//---------------------------------------------------------------------------------------------------------------
//
//  HAUD 2024.12.19
//
//
//  fb_SenderBuffer
//  - inherits fb_Instance, which provides a design pattern in order to build different specific processes in a structured way
//  - uses 1 XtsStation via _ItfProcessCollector
//  - used for targeting movers to predetermined substation of process control (one to one)
//  - processes are connected via linked list
//    - entry in list is detected
//    - entry in list determines count and place of used XtsStations in target process
//
//
//  - constructed with fb_Instance main state (_eState) in addition to a substate (_eStateProgress)
//  - substate enables to handle procedures within main state by preventing race conditions 
//    with the help of small steps and decisions with clear separation from each other 
//
//---------------------------------------------------------------------------------------------------------------//
// This SOFTWARE is provided as an Exemple by THE PROVIDER "as is" and "with all faults." THE PROVIDER makes no  //
// representations or warranties of any kind concerning the safety, suitability, lack of viruses, inaccuracies,  //
// typographical errors, or other harmful components of this SOFTWARE. There are inherent dangers in the use of  //
// any software, and you are solely responsible for determining whether this SOFTWARE is compatible with your    //
// equipment and other software installed on your equipment. You are also solely responsible for the protection  //
// of your equipment and backup of your data, and THE PROVIDER will not be liable for any damages you may suffer //
// in connection with using, modifying, or distributing this SOFTWARE.                                           //
//---------------------------------------------------------------------------------------------------------------//
FUNCTION_BLOCK fb_SenderBuffer EXTENDS fb_Instance
VAR
  _nProcessTarget               : E_INSTANCE;     // who am I connected to

  // target XTS station range
  _nTargetStationLast           : UINT;           // where does the target process end
  _nTargetStationFirst          : UINT;           // where does the target process start

  _rCheckPos                    : LREAL;

  _WriteResult                  : ST_PROCESS_LIST_RESULT;   // last job written to target
  _DeleteResult                 : ST_PROCESS_LIST_RESULT;   // last job executed

  _idx                          : UINT;
  _nTargetIndex                 : ARRAY[1..SIZEOF(T_PROCESS)*8] OF USINT; // helper var to copy to my process (_ItfProcessCollector[_nProcess].TargetIndex)

  _MoverInfo                    : ST_MOVER_INFO;      // Information from the Mover in Station
  _StationState                 : ST_STATION_STATE;   // fb_SenderBufferInfeed has only one XtsStation to work

  _nBatch                       : udint;
END_VAR

//-----------------------------------------------------------------------------
//-----------------------------------------------------------------------------
// check pointer and interface
// connect Ctrl/State to _ItfProcessCollector
// set message device identification
//-----------------------------------------------------------------------------
IF NOT Check() THEN 
  RETURN; 
END_IF
//-----------------------------------------------------------------------------
// check init command (hard reset)
//-----------------------------------------------------------------------------
_eCmd                                 := _InstanceCtrl[_nProcess].Cmd;
IF (_eCmd <> _eCmdOld)
THEN
  CASE _eCmd
  OF
    E_INSTANCE_CMD.INIT:
      // clear init info
      _nBatch                         := 0;
      _eInit                          := _ItfProcessCollector[_nProcess].Init(FALSE);
  
      IF _ItfProcessList[_nProcess].InitList()  // clear linked list
      THEN
        Clear();
        _eStateInstance               := E_INSTANCE_STATE.INIT;
        _eStateProgress               := E_PROGRESS.PROGRESS_INIT;
      END_IF

    E_INSTANCE_CMD.CLEAR:
        _eStateInstance               := E_INSTANCE_STATE.DISABLED;
        _eStateProgress               := E_PROGRESS.PROGRESS_INIT;
  END_CASE
  CmdLog();
  _eCmdOld                            := _eCmd;
END_IF
//-----------------------------------------------------------------------------
// cyclic information of mover and station
//-----------------------------------------------------------------------------
_StationState                         := _ItfProcessCollector[_nProcess].GetStationState  (_ItfProcessCollector[_nProcess].StationLast);
_MoverInfo                            := _ItfProcessCollector[_nProcess].GetMoverInStation(_ItfProcessCollector[_nProcess].StationLast);
//-----------------------------------------------------------------------------
//-----------------------------------------------------------------------------
// state machine for buffer to OutputR1 and OutputR2
//-----------------------------------------------------------------------------
CASE _eStateInstance // main state machine
OF
  E_INSTANCE_STATE.NULL:           // first cycle init
    IF _ItfProcessList[_nProcess].InitList()
    THEN
      _eInit                          := _ItfProcessCollector[_nProcess].Init(FALSE);
      _eStateProgress                 := E_PROGRESS.PROGRESS_INIT;
      _eStateInstance                 := E_INSTANCE_STATE.INIT;
    END_IF


  E_INSTANCE_STATE.INIT:              // plausibility checks and _ItfProcessCollector Init
    //-------------------------------------------------------------------------
    CASE _eStateProgress
    OF
    //-------------------------------------------------------------------------
      E_PROGRESS.PROGRESS_ERROR:
        IF (_nProcessTarget > 0) AND
           (_nProcessTarget < E_INSTANCE.INSTANCE_MAX)
        THEN
          _eStateProgress             := E_PROGRESS.PROGRESS_INIT;
        END_IF

    // E_INSTANCE_STATE.INIT:
    //-------------------------------------------------------------------------
      E_PROGRESS.PROGRESS_INIT:
        IF NOT (_nProcessTarget > 0) OR
           NOT (_nProcessTarget < E_INSTANCE.INSTANCE_MAX)
        THEN
          // an invalid target you must have not
          _eStateProgress             := E_PROGRESS.PROGRESS_ERROR;
        ELSE
          _eStateProgress             := E_PROGRESS.PROGRESS_BUSY;
        END_IF

    // E_INSTANCE_STATE.INIT:
    //-------------------------------------------------------------------------
      E_PROGRESS.PROGRESS_BUSY:
        // wait for my process collector check (_State.Check) to be done
        //  - checks range of XtsStations
        //  - checks count of XtsStations
        IF (_State.Check = E_PROCESS_CHECK.PROCESS_CHECK_DONE)
        THEN
          _eInit                      := _ItfProcessCollector[_nProcess].Init(TRUE);
  
          IF (_eInit = E_PROGRESS.PROGRESS_DONE)
          THEN
            IF NOT (_nProcessTarget > 0) OR
               NOT (_nProcessTarget < E_INSTANCE.INSTANCE_MAX)
            THEN
              // an invalid target you must have not
              _eStateProgress         := E_PROGRESS.PROGRESS_ERROR;

              _stMsg.eType            := E_MessageType.eMessageError;
              _stMsg.eSubdevice       := e_Subdevice.Instance_BufferOutfeed;
              _stMsg.iErrorNumber     := _nProcessTarget;
              _stMsg.sText            := concat(TO_STRING(_eStateInstance), ': ProcessTarget: ');
              _stMsg.sText            := concat(_stMsg.sText, TO_STRING(_eStateProgress));
              f_MessageSet(_stMsg);

            ELSE
              _nTargetStationLast     := _ItfProcessCollector[_nProcessTarget].StationLast;
              _nTargetStationFirst    := _ItfProcessCollector[_nProcessTarget].StationFirst;

              // initialization of Infeed: _ItfProcessCollector with XtsStation
              _Ctrl.Cmd               := E_PROCESS_CTRL.PROCESS_DISABLE;  // first, switch off _ItfProcessCollector and XtsStation
              _eStateProgress         := E_PROGRESS.PROGRESS_INIT;        // clear sub state
              _eStateInstance         := E_INSTANCE_STATE.DISABLED;       // switch to disabled as default after startup
            END_IF
          END_IF
        END_IF
    END_CASE
END_CASE
//-----------------------------------------------------------------------------
//-----------------------------------------------------------------------------
// DISABLED:
//  - clear local list result data
//  - wait for enable from the outside
//  - wait for an entry in my list
//-----------------------------------------------------------------------------
CASE _eStateInstance
OF
  E_INSTANCE_STATE.DISABLED:
    //-------------------------------------------------------------------------
    CASE _eStateProgress
    OF
      E_PROGRESS.PROGRESS_INIT:
        _eStateProgress               := E_PROGRESS.PROGRESS_BUSY;
        // clear data for a new round
        memset(ADR(_ListResult), 0, SIZEOF(_ListResult));

        _Ctrl.ActivateStation         := 0;
        _Ctrl.NestMask                := 1;
        
    // E_INSTANCE_STATE.DISABLED:
    //-------------------------------------------------------------------------
      E_PROGRESS.PROGRESS_BUSY:
        CASE _eCmd
        OF
          E_INSTANCE_CMD.ENABLE:      // turn it on!!
            _eStateInstance           := E_INSTANCE_STATE.DETECTION;
            _eStateProgress           := E_PROGRESS.PROGRESS_BUSY;

  
            IF (_MessageLevel > E_MessageType.eMessageInfo)
            THEN
              _stMsg.eType            := E_MessageType.eMessageVerbose;
              _stMsg.eSubdevice       := e_Subdevice.Instance_Sender_Buffer;
              _stMsg.iErrorNumber     := 0;
              _stMsg.sText            := concat(TO_STRING(_eStateInstance), ': ');
              _stMsg.sText            := concat(_stMsg.sText, TO_STRING(_eStateProgress));
              f_MessageSet(_stMsg);
            END_IF
        END_CASE
    END_CASE
END_CASE
//-----------------------------------------------------------------------------
// DETECTION: 
//  - check inked list and GetHead()
//  - copy job data
//  - switch on process
//-----------------------------------------------------------------------------
CASE _eStateInstance
OF
  E_INSTANCE_STATE.DETECTION:
    //-------------------------------------------------------------------------
    CASE _eStateProgress
    OF
      E_PROGRESS.PROGRESS_INIT:
        IF (_eCmd = E_INSTANCE_CMD.PROCEED)
        THEN
          _eStateProgress             := E_PROGRESS.PROGRESS_BUSY;
        END_IF
    END_CASE
    // E_INSTANCE_STATE.DETECTION
    //-------------------------------------------------------------------------
    CASE _eStateProgress
    OF
      E_PROGRESS.PROGRESS_BUSY:
        IF (_eCmd = E_INSTANCE_CMD.DISABLE)
        THEN
          _eStateInstance             := E_INSTANCE_STATE.DISABLED;
          _eStateProgress             := E_PROGRESS.PROGRESS_INIT;

        ELSIF (_ItfProcessList[_nProcess].Count > 0)
        THEN
          // get new job order for my process
          // check my list for a new round of movers
          _ListResult                 := _ItfProcessList[_nProcess].GetHead();  // the list results carries information about the requirements of the target process (who and where)

          IF (_ListResult.wState <> 0)
          THEN
            // error in list results must not appear
            // if you land here, there is somethng wrong with the initialization or configuration of the linked list
            _eStateProgress           := E_PROGRESS.PROGRESS_ERROR;

            _stMsg.eType              := E_MessageType.eMessageError;
            _stMsg.eSubdevice         := e_Subdevice.Process_LinkedList_GetHead;
            _stMsg.iErrorNumber       := _ListResult.wState;
            _stMsg.sText              := concat(TO_STRING(_eStateInstance), ': ');
            _stMsg.sText              := concat(_stMsg.sText, TO_STRING(_eStateProgress));
            f_MessageSet(_stMsg);

          ELSE
            IF (_MessageLevel > E_MessageType.eMessageError)
            THEN
              _stMsg.eType            := E_MessageType.eMessageInfo;
              _stMsg.eSubdevice       := e_Subdevice.Process_LinkedList_GetHead;
              _stMsg.iErrorNumber     := 0;
              _stMsg.sText            := concat(TO_STRING(_eStateInstance), ': ');
              _stMsg.sText            := concat(_stMsg.sText, '_ListResult.stData.wTarget: ');
              _stMsg.sText            := concat(_stMsg.sText, _ItfProcessCollector[_nProcess].BitsToString(_ListResult.stData.wTarget));
              f_MessageSet(_stMsg);
            END_IF

            _ProcessData              := _ListResult.stData;  // list result contains data for target process

            IF NOT (_ProcessData.wTarget > 0)
            THEN
              // no data, no cry
              _DeleteResult           := _ItfProcessList[_nProcess].RemoveHeadValue();
            ELSE
              _eStateProgress         := E_PROGRESS.PROGRESS_CHECK;

              IF (_MessageLevel > E_MessageType.eMessageEmpty)
              THEN
                _stMsg.eType            := E_MessageType.eMessageBatch;
                _stMsg.eSubdevice       := e_Subdevice.Instance_Sender_Buffer;
                _stMsg.iErrorNumber     := _ProcessData.wTarget;
                _stMsg.sText            := concat('_ProcessData.wTarget: ', _ItfProcessCollector[_nProcess].BitsToString(_ProcessData.wTarget));
                _stMsg.sText            := concat(_stMsg.sText, ': ');
                _stMsg.sText            := concat(_stMsg.sText, TO_STRING(_eStateProgress));
                _stMsg.sText            := concat(_stMsg.sText, ': ');
                _stMsg.sText            := concat(_stMsg.sText, TO_STRING(e_message_batch.MSG_BATCH_JOB_STARTED));
                f_MessageSet(_stMsg);
              END_IF
            END_IF

            // check target mask for entries
            IF NOT (_ProcessData.wTarget > 0)
            THEN
              //_eStateProgress         := E_PROGRESS.PROGRESS_ERROR;

              _stMsg.eType            := E_MessageType.eMessageWarning;
              _stMsg.eSubdevice       := e_Subdevice.Process_LinkedList_CheckData;
              _stMsg.iErrorNumber     := 666;
              _stMsg.sText            := concat(TO_STRING(_eStateInstance), ': ');
              _stMsg.sText            := concat(_stMsg.sText, '_ProcessData.wTarget: ');
              _stMsg.sText            := concat(_stMsg.sText, _ItfProcessCollector[_nProcess].BitsToString(_ProcessData.wTarget));
              f_MessageSet(_stMsg);
            END_IF
          END_IF
        END_IF
    END_CASE
    // E_INSTANCE_STATE.DETECTION
    //-------------------------------------------------------------------------
    CASE _eStateProgress
    OF
      E_PROGRESS.PROGRESS_CHECK:
        // check for disabled process interface state
        CASE _State.State
        OF
          E_PROCESS_STATE.PROCESS_DISABLE:

          CASE _State.Result
          OF
            E_PROGRESS.PROGRESS_BUSY:     // busy from _State.Result means, waiting for input
              // now the preparation for the target process may begin
              _Ctrl.Cmd               := E_PROCESS_CTRL.PROCESS_ENABLE;
              _Ctrl.ActivateStation   := 1; // I am a sender, there is only one XtsStation to work

              _eStateInstance         := E_INSTANCE_STATE.ENABLED;      // go check if my process is switched on
              _eStateProgress         := E_PROGRESS.PROGRESS_INIT;      // reset substate

              IF (_MessageLevel > E_MessageType.eMessageInfo)
              THEN
                _stMsg.eType          := E_MessageType.eMessageVerbose;
                _stMsg.eSubdevice     := e_Subdevice.Instance_Sender_Buffer;
                _stMsg.iErrorNumber   := 0;
                _stMsg.sText          := concat(TO_STRING(_eStateInstance), ': ');
                _stMsg.sText          := concat(_stMsg.sText, TO_STRING(_eStateProgress));
                _stMsg.sText          := concat(_stMsg.sText, ': ');
                _stMsg.sText          := concat(_stMsg.sText, TO_STRING(_Ctrl.Cmd));
                f_MessageSet(_stMsg);
              END_IF
          END_CASE
        END_CASE
    END_CASE
END_CASE
//-----------------------------------------------------------------------------
// ENABLED
//  - check process for enabled station
//  - switch to infeed
//  - check if infeed is active
//  - allow movers to enter
//-----------------------------------------------------------------------------
CASE _eStateInstance
OF
  E_INSTANCE_STATE.ENABLED:
    //-------------------------------------------------------------------------
    CASE _eStateProgress
    OF
      E_PROGRESS.PROGRESS_INIT:
        CASE _State.State
        OF
          E_PROCESS_STATE.PROCESS_ENABLE:
          CASE _State.Result
          OF
            E_PROGRESS.PROGRESS_BUSY:
              // now my process and all XtsStations within are switched on
              // check infeed into my process
              _Ctrl.Cmd               := E_PROCESS_CTRL.PROCESS_STATIONS_INFEED; // tells my process to go check the infeed
              _eStateProgress         := E_PROGRESS.PROGRESS_BUSY; // go check how the infeed into my process is doing

              IF (_MessageLevel > E_MessageType.eMessageInfo)
              THEN
                _stMsg.eType          := E_MessageType.eMessageVerbose;
                _stMsg.eSubdevice     := e_Subdevice.Instance_Sender_Buffer;
                _stMsg.iErrorNumber   := 0;
                _stMsg.sText          := concat(TO_STRING(_eStateInstance), ': ');
                _stMsg.sText          := concat(_stMsg.sText, TO_STRING(_eStateProgress));
                f_MessageSet(_stMsg);
              END_IF
          END_CASE
        END_CASE
    END_CASE
    // E_INSTANCE_STATE.ENABLED:
    //-------------------------------------------------------------------------
    CASE _eStateProgress
    OF
      E_PROGRESS.PROGRESS_BUSY:
        CASE _State.State
        OF
          E_PROCESS_STATE.PROCESS_STATIONS_INFEED:
          CASE _State.Result
          OF
            E_PROGRESS.PROGRESS_BUSY:
              // now we know who wants to enter
              _Ctrl.Cmd               := E_PROCESS_CTRL.PROCESS_STATIONS_SEND;  // send mover to outfeed process
              _eStateProgress         := E_PROGRESS.PROGRESS_PREPARE;           // go check sending of mover
  
              IF (_MessageLevel > E_MessageType.eMessageInfo)
              THEN
                _stMsg.eType          := E_MessageType.eMessageVerbose;
                _stMsg.eSubdevice     := e_Subdevice.Instance_Sender_Buffer;
                _stMsg.iErrorNumber   := 0;
                _stMsg.sText          := concat(TO_STRING(_Ctrl.Cmd), ': ');
                _stMsg.sText          := concat(_stMsg.sText, TO_STRING(_eStateProgress));
                f_MessageSet(_stMsg);
  
                _stMsg.eType          := E_MessageType.eMessageVerbose;
                _stMsg.eSubdevice     := e_Subdevice.Instance_Sender_Buffer;
                _stMsg.iErrorNumber   := 0;
                _stMsg.sText          := concat(TO_STRING(_eStateInstance), ': ');
                _stMsg.sText          := concat(_stMsg.sText, TO_STRING(_eStateProgress));
                f_MessageSet(_stMsg);
              END_IF
          END_CASE
        END_CASE
    END_CASE
    // E_INSTANCE_STATE.ENABLED:
    //-------------------------------------------------------------------------
    CASE _eStateProgress
    OF
      E_PROGRESS.PROGRESS_PREPARE:
        CASE _State.State
        OF
          E_PROCESS_STATE.PROCESS_STATIONS_OUTFEED:
          CASE _State.Result
          OF
            E_PROGRESS.PROGRESS_BUSY:
              IF (_MoverInfo.rModuloActPos > _rCheckPos)
              THEN
                // mover is in range and can leave now
                _eStateInstance       := E_INSTANCE_STATE.FINISH;     // go send mover
                _eStateProgress       := E_PROGRESS.PROGRESS_INIT;    // reset substate
  
                IF (_MessageLevel > E_MessageType.eMessageError)
                THEN
                  _stMsg.eType        := E_MessageType.eMessageInfo;
                  _stMsg.eSubdevice   := e_Subdevice.Instance_Sender_Buffer;
                  _stMsg.iErrorNumber := _StationState.nMoverId;
                  _stMsg.sText        := concat(TO_STRING(_eStateInstance), ': ');
                  _stMsg.sText        := concat(_stMsg.sText, TO_STRING(_eStateProgress));
                  f_MessageSet(_stMsg);
                END_IF
              END_IF
          END_CASE
        END_CASE
    END_CASE
END_CASE
//-----------------------------------------------------------------------------
// FINISH:
//  - write target (OutputR2 and OutputR1)
//  - command outfeed of mover
//  - AddTail() at TargetProcess
//  - check to proceed
//-----------------------------------------------------------------------------
CASE _eStateInstance
OF
  E_INSTANCE_STATE.FINISH:
    //-------------------------------------------------------------------------
    CASE _eStateProgress
    OF
      E_PROGRESS.PROGRESS_INIT:
      _eStateProgress                 := E_PROGRESS.PROGRESS_BUSY;

      // the sending of mover
      // many movers to one target
      _nTargetIndex[1]                := TO_USINT(_nTargetStationLast);

      _ItfProcessCollector[_nProcess].TargetIndex := _nTargetIndex; // write Xts target onto my ProcessCollector interface

      FOR _idx := 1 TO (SIZEOF(T_PROCESS)*8)
      DO
        IF (_ItfProcessCollector[_nProcess].BitGet(_ProcessData.wTarget, _idx-1))
        THEN
          IF (_MessageLevel > E_MessageType.eMessageVerbose)
          THEN
            _stMsg.eType              := E_MessageType.eMessageSentient;
            _stMsg.eSubdevice         := e_Subdevice.Instance_Sender_Buffer;
            _stMsg.iErrorNumber       := _idx;
            _stMsg.sText              := concat('I_AM _ProcessData.wTarget: ', 
                                         _ItfProcessCollector[_nProcess].BitsToString(_ProcessData.wTarget));
            f_MessageSet(_stMsg);
          END_IF

          _ProcessData.wTarget        := _ItfProcessCollector[_nProcess].
                                         BitDel(_ProcessData.wTarget, _idx-1);

          IF (_MessageLevel > E_MessageType.eMessageVerbose)
          THEN
            _stMsg.eType              := E_MessageType.eMessageSentient;
            _stMsg.eSubdevice         := e_Subdevice.Instance_Sender_Buffer;
            _stMsg.iErrorNumber       := _idx;
            _stMsg.sText              := concat('I_WAS _ProcessData.wTarget: ', 
                                         _ItfProcessCollector[_nProcess].BitsToString(_ProcessData.wTarget));
            f_MessageSet(_stMsg);
          END_IF
          EXIT;
        END_IF
      END_FOR
    END_CASE
    //-------------------------------------------------------------------------
    CASE _eStateProgress
    OF
      E_PROGRESS.PROGRESS_BUSY:
        CASE _State.State
        OF
          E_PROCESS_STATE.PROCESS_STATIONS_OUTFEED: // check my process' state
          CASE _State.Result
          OF
            E_PROGRESS.PROGRESS_BUSY:
            // now data is prepared and copied to the right places
            CASE _eCmd
            OF
              E_INSTANCE_CMD.FINISH:      // send mover out!!
                _Ctrl.Cmd             := E_PROCESS_CTRL.PROCESS_STATIONS_OUTFEED; // release the kraken!

                IF (_ProcessData.wTarget = 0)
                THEN
                  // all done, go check for new list entry 
                  _nBatch             := _nBatch + 1;
                  _eStateProgress     := E_PROGRESS.PROGRESS_DONE;                // mover is on its way
                  _stMsg.iErrorNumber := 0;

                  IF (_MessageLevel > E_MessageType.eMessageVerbose)
                  THEN
                    _stMsg.eType              := E_MessageType.eMessageSentient;
                    _stMsg.eSubdevice         := e_Subdevice.Instance_Sender_Buffer;
                    _stMsg.iErrorNumber       := 0;
                    _stMsg.sText              := concat('I_GONE _ProcessData.wTarget: ', 
                                                 _ItfProcessCollector[_nProcess].BitsToString(_ProcessData.wTarget));
                    f_MessageSet(_stMsg);
                  END_IF
                  IF (_MessageLevel > E_MessageType.eMessageEmpty)
                  THEN
                    _stMsg.eType        := E_MessageType.eMessageBatch;
                    _stMsg.eSubdevice   := e_Subdevice.Instance_Outfeed;
                    _stMsg.iErrorNumber := 0;
                    _stMsg.sText        := concat(TO_STRING(_eStateProgress), ': ');
                    _stMsg.sText        := concat(_stMsg.sText, TO_STRING(e_message_batch.MSG_BATCH_JOB_DONE));
                    f_MessageSet(_stMsg);
                  END_IF
                ELSE
                  // job not done
                  _eStateProgress     := E_PROGRESS.PROGRESS_PREPARE;
                  IF (_MessageLevel > E_MessageType.eMessageVerbose)
                  THEN
                    _stMsg.eType              := E_MessageType.eMessageSentient;
                    _stMsg.eSubdevice         := e_Subdevice.Instance_Sender_Buffer;
                    _stMsg.iErrorNumber       := 0;
                    _stMsg.sText              := concat('I_RETURN _ProcessData.wTarget: ', 
                                                 _ItfProcessCollector[_nProcess].BitsToString(_ProcessData.wTarget));
                    f_MessageSet(_stMsg);
                  END_IF
                  IF (_MessageLevel > E_MessageType.eMessageEmpty)
                  THEN
                    _stMsg.eType        := E_MessageType.eMessageBatch;
                    _stMsg.eSubdevice   := e_Subdevice.Instance_Outfeed;
                    _stMsg.iErrorNumber := 0;
                    _stMsg.sText        := concat(TO_STRING(_eStateProgress), ': ');
                    _stMsg.sText        := concat(_stMsg.sText, TO_STRING(e_message_batch.MSG_BATCH_NEXT_IN_JOB));
                    f_MessageSet(_stMsg);
                  END_IF
                END_IF
            END_CASE
          END_CASE
        END_CASE
    END_CASE
    //-------------------------------------------------------------------------
    CASE _eStateProgress
    OF
      E_PROGRESS.PROGRESS_PREPARE:
        CASE _State.State
        OF
          E_PROCESS_STATE.PROCESS_DISABLE: // check my process' state
          CASE _State.Result
          OF
            E_PROGRESS.PROGRESS_BUSY:
              _Ctrl.Cmd                     := E_PROCESS_CTRL.PROCESS_ENABLE;
              _eStateInstance               := E_INSTANCE_STATE.ENABLED;
              _eStateProgress               := E_PROGRESS.PROGRESS_INIT;
          END_CASE
        END_CASE
    END_CASE
    //-------------------------------------------------------------------------
    CASE _eStateProgress
    OF
      E_PROGRESS.PROGRESS_DONE:
        CASE _State.State
        OF
          E_PROCESS_STATE.PROCESS_DISABLE: // check my process' state
          CASE _State.Result
          OF
            E_PROGRESS.PROGRESS_BUSY:
              _DeleteResult                 := _ItfProcessList[_nProcess].RemoveHeadValue();
              IF (_DeleteResult.wState <> 0)
              THEN
                _eStateProgress             := E_PROGRESS.PROGRESS_ERROR;
              ELSE
                IF (_MessageLevel > E_MessageType.eMessageError)
                THEN
                  _stMsg.eType        := E_MessageType.eMessageInfo;
                  _stMsg.eSubdevice   := e_Subdevice.Process_LinkedList_RemoveHead;
                  _stMsg.iErrorNumber := 0;
                  _stMsg.sText        := concat(TO_STRING(_eStateInstance), ': ');
                  _stMsg.sText        := concat(_stMsg.sText, TO_STRING(_eStateProgress));
                  f_MessageSet(_stMsg);
                END_IF

                _eStateInstance             := E_INSTANCE_STATE.DISABLED;
                _eStateProgress             := E_PROGRESS.PROGRESS_INIT;
              END_IF
          END_CASE
        END_CASE
    END_CASE
END_CASE
//-----------------------------------------------------------------------------
//-----------------------------------------------------------------------------
_InstanceState[_nProcess].State       := _eStateInstance;
_InstanceState[_nProcess].Progress    := _eStateProgress;

PROPERTY CheckPosition : lreal
GET
CheckPosition := _rCheckPos;
END_GET
SET
_rCheckPos := CheckPosition;
END_SET
END_PROPERTY

METHOD Clear : BOOL
VAR_INPUT
END_VAR
memset(ADR(_nTargetIndex), 0, SIZEOF(_nTargetIndex));

//_eStateInstance                         := E_INSTANCE_STATE.DISABLED;
_eStateProgress                 := E_PROGRESS.PROGRESS_INIT;

Clear                           := TRUE;
END_METHOD

PROPERTY ProcessTarget : E_INSTANCE
GET
ProcessTarget := _nProcessTarget;
END_GET
SET
_nProcessTarget := ProcessTarget;
END_SET
END_PROPERTY

END_FUNCTION_BLOCK

(* stored: Version 1.1.0.1, ProductVersion 3.1.4026.13
   POU fb_SenderBuffer: Id {0c3bbcb7-2e32-448d-927f-70f07eaaefdd}, SpecialFunc None
   Property CheckPosition: Id {81019363-a4f7-41e9-a92f-706b94c041bc}
   Get Get: Id {3ca52888-1831-4fb8-bfad-b16c9277def2}
   Set Set: Id {bac3b342-2cbe-4417-b6f8-5ba191d6a576}
   Method Clear: Id {f2d37d2f-3514-4055-adbd-e2ca4cba26e1}
   Property ProcessTarget: Id {46172c2c-8935-49f5-ab70-cd18f4abacc0}
   Get Get: Id {dde22dda-2d7e-408f-9b09-a81a080d2f99}
   Set Set: Id {c4c8f051-cf85-47f1-999c-91dbb3eeb3de} *)
